# EPICS substitutions: db/music_hv.substitutions
file "db/music_hv.template"
{
    pattern { FC, CH }
            { 1,  0  }
            { 2,  1  }
            { 3,  2  }
            { 4,  3  }
}
